FUNCTION_BLOCK System_AppInfo
VAR_INPUT
	
END_VAR
VAR_OUTPUT
	ObjectID: UDINT;
	TaskCount: UDINT;
	OnlineChangeCount: UDINT;
	Flags: DWORD;
	AdsPort: UINT;
	BootDataLoaded: BOOL;
	OldBootData: BOOL;
	AppTimestamp: DATE_AND_TIME;
	KeepOutputsOnBreakpoint: BOOL;
	ShutdownInProgress: BOOL;
	LicensePending: BOOL;
	BlueScreenOccured: BOOL;
	LoggedIn: BOOL;
	PersistentStatus: EPlcPersistentStatus;
	TcComSrvPointer: ITComObjectServer;
	AppName: STRING(63);
	ProjectName: STRING(63);
END_VAR
VAR
	(* AppInfo Source Data *)
	_ThisAppInfo: PlcAppSystemInfo;
	
END_VAR

_ThisAppInfo := TwinCAT_SystemInfoVarList._AppInfo;
ObjectID := _ThisAppInfo.ObjId;
TaskCount := _ThisAppInfo.TaskCnt;
OnlineChangeCount := _ThisAppInfo.OnlineChangeCnt;
Flags := _ThisAppInfo.Flags;
AdsPort := _ThisAppInfo.AdsPort;
BootDataLoaded := _ThisAppInfo.BootDataLoaded;
OldBootData := _ThisAppInfo.OldBootData;
AppTimestamp := _ThisAppInfo.AppTimestamp;
KeepOutputsOnBreakpoint := _ThisAppInfo.KeepOutputsOnBP;
ShutdownInProgress := _ThisAppInfo.ShutdownInProgress;
LicensePending := _ThisAppInfo.LicensesPending;
BlueScreenOccured := _ThisAppInfo.BSODOccured;
LoggedIn := _ThisAppInfo.LoggedIn;
PersistentStatus := _ThisAppInfo.PersistentStatus;
TcComSrvPointer := _ThisAppInfo.TComSrvPtr;
AppName := _ThisAppInfo.AppName;
ProjectName := _ThisAppInfo.ProjectName;

END_FUNCTION_BLOCK

(* stored: Version 1.1.0.1, ProductVersion 3.1.4024.12
   POU System_AppInfo: Id {d5dba280-0c9e-480e-abc1-3ad6d934ba13}, SpecialFunc None *)
